// TIA Portal V20 export
// export: Created 2025-12-01T14:57:43.7289768Z, ExportSetting None, DisplayName Totally Integrated Automation Portal, DisplayVersion V20 Update 3, DisplayName TIA Portal Openness, DisplayVersion V20 Update 3, DisplayName TIA Portal Version Control Interface, DisplayVersion V20 Update 3, DisplayName STEP 7 Professional, DisplayVersion V20 Update 3, DisplayName STEP 7 Safety, DisplayVersion V20 Update 2, DisplayName WinCC Basic/Comfort/Advanced, DisplayVersion V20 Update 3, DisplayName WinCC Professional, DisplayVersion V20 Update 3, DisplayName WinCC Unified, DisplayVersion V20 Update 3
FUNCTION "FC512_TL_EtiquetaLeida_EnMesa_ULINT" : Void   // FC512, LAD
{ S7_Optimized_Access := 'FALSE' }
AUTHOR : T_LIGERO
NAME : 20141014
VERSION : 4.0
// stored: AutoNumber false, SetENOAutomatically false
   VAR_INPUT
      Mesa : UInt;   // Numero de Mesa CON OFFSET
      NumSCR : UInt;   // Numero de Scanner asociada a la mesa
      LongFIFO_SCR : UInt;   // Numero de Lecturas que se pueden Almacenar
      MesaDeJDT02 : Bool;
   END_VAR
   VAR_TEMP
      Datos_scanner : "ROUT_Orden_Fifo_Scanner";
      codigo_string : String[20];
      mesa_string : String[5];
      i : Int;
      FIFO_OK : Bool;
      longitud : Int;
      posicion : Int;
   END_VAR
BEGIN

REGION Network 1 (SCL): escribir los datos en el string
   "FC571_Leer_Datos_Fifo"(DB_FIFO_Ordenes:="ROUT_NDB_FIFO_Odr_SCR",
                           Num_Scanner:=#NumSCR,
                           Long_FIFO:=#LongFIFO_SCR,
                           Posicion_FIFO:=1,
                           Datos_Scanner_Cruce=>#Datos_scanner);

   IF #Datos_scanner.Orden = 0 THEN
       RETURN;
   END_IF;




   // MIRAR SI TENEMOS ESPACIO PARA EMITIR EL MENSAJE ANTES DE FORMATEARLO
   IF #MesaDeJDT02 = true THEN
       REGION buscar en JDT2

           #posicion := -1;
           FOR #i := 0 TO 100 BY 1 DO
               #longitud := LEN("DB197_eventos_generados_routing_JDT2".evento[#i]);
               IF #longitud = 0 THEN
                   #posicion := #i;
                   EXIT;
               END_IF;
           END_FOR;

           // si no hay sitio para escribir salimos del bloque
           IF #posicion = -1 THEN
               RETURN;
           END_IF;
       END_REGION
       ;
   ELSE
       REGION buscar en JDT1

           #posicion := -1;
           FOR #i := 0 TO 100 BY 1 DO
               #longitud := LEN("DB198_eventos_generados_routing_JDT1".evento[#i]);
               IF #longitud = 0 THEN
                   #posicion := #i;
                   EXIT;
               END_IF;
           END_FOR;

           // si no hay sitio para escribir salimos del bloque
           IF #posicion = -1 THEN
               RETURN;
           END_IF;
       END_REGION
   END_IF;
   // buscamos hueco en el db donde vamos a escribir los eventos antes de empezar la conversión
   // 

   // si hay sitio para convertir iniciamos la conversión de los parametros a enviar en el mensaje

   #mesa_string :=  DELETE(IN := (UINT_TO_STRING(IN := #Mesa)), L := 1, P := 1);
   #codigo_string := DELETE(IN := (ULINT_TO_STRING(IN := #Datos_scanner.Identificador)), L := 1, P := 1);

   // concatenamos el mensaje 
   // 
   IF #MesaDeJDT02 = true THEN

       "DB197_eventos_generados_routing_JDT2".evento[#posicion] := CONCAT(IN1 := '{PRES[MESA]', IN2 := #mesa_string, IN3 := '[SSCC]', IN4 := #codigo_string, IN5 := '[MOTI]NORM', IN6 :="DB921_DATOS_FECHA_HORA".TIME_STAMP , IN7:='}');

       ELSE
           "DB198_eventos_generados_routing_JDT1".evento[#posicion] := CONCAT(IN1 := '{PRES[MESA]', IN2 := #mesa_string, IN3 := '[SSCC]', IN4 := #codigo_string, IN5 := '[MOTI]NORM', IN6 :="DB921_DATOS_FECHA_HORA".TIME_STAMP , IN7:='}');

   END_IF;

       "FC502_Actualiza_FIFO_SCR"(DB_FIFO_Ordenes:="ROUT_NDB_FIFO_Odr_SCR",
                                  Num_Scanner:=#NumSCR,
                                  Long_FIFO:=#LongFIFO_SCR,
                                  FIFO_OK:=#FIFO_OK);
END_REGION
END_FUNCTION
